(* IEC 61131-3 sources: RL_MAR/experiments/comparison/llm4plc/results/deepseek-ai-DeepSeek-V3.2_20260506_104945/20260506_124638, 3 files *)

(* ---- generated_code_iteration_0.st ---- *)
START_ST
FUNCTION_BLOCK CapsuleFillingMachineControl
VAR_INPUT
    CapsuleWeight : REAL;
    TargetWeight : REAL;
    CapsuleInPosition : BOOL;
    HopperEmpty : BOOL;
END_VAR
VAR_OUTPUT
    FeederMotor : BOOL;
    FillingMotor : BOOL;
    ConveyorMotor : BOOL;
    FillingInProgress : BOOL;
    ErrorFlag : BOOL;
    FillingTimeoutError : BOOL;
    CapsuleDetectionError : BOOL;
END_VAR
VAR
    state : INT;
    prevState : INT;
    fillingTimer : TON;
    conveyingTimer : TON;
    capsuleDetectionTimer : TON;
    tolerance : REAL := 0.1;
    conveyingTime : TIME := T#2s;
    fillingTimeout : TIME := T#10s;
    detectionTimeout : TIME := T#5s;
    pidController : PID;
    pidSetpoint : REAL;
    pidInput : REAL;
    pidOutput : REAL;
    pidKp : REAL := 1.0;
    pidKi : REAL := 0.1;
    pidKd : REAL := 0.05;
    manualReset : BOOL;
END_VAR

(* Safety Check - Immediate Override *)
IF HopperEmpty THEN
    FeederMotor := FALSE;
    FillingMotor := FALSE;
    ConveyorMotor := FALSE;
    FillingInProgress := FALSE;
    state := 4; (* ERROR state *)
    RETURN;
END_IF;

(* Weight Validation - Immediate Override *)
IF CapsuleWeight >= TargetWeight THEN
    FeederMotor := FALSE;
    FillingMotor := FALSE;
    ConveyorMotor := FALSE;
    FillingInProgress := FALSE;
    state := 4; (* ERROR state *)
    RETURN;
END_IF;

(* Main State Machine *)
CASE state OF
    0: (* IDLE *)
        FeederMotor := TRUE; (* Assumption: Feeder ON when not empty *)
        FillingMotor := FALSE;
        ConveyorMotor := FALSE;
        FillingInProgress := FALSE;
        ErrorFlag := FALSE;
        FillingTimeoutError := FALSE;
        CapsuleDetectionError := FALSE;

        capsuleDetectionTimer(IN:=FALSE, PT:=detectionTimeout);

        IF CapsuleInPosition AND (CapsuleWeight < TargetWeight) THEN
            state := 1; (* CONVEYING *)
            conveyingTimer(IN:=TRUE, PT:=conveyingTime);
        END_IF;

    1: (* CONVEYING *)
        FeederMotor := TRUE;
        FillingMotor := FALSE;
        ConveyorMotor := TRUE;
        FillingInProgress := FALSE;

        capsuleDetectionTimer(IN:=TRUE, PT:=detectionTimeout);

        (* Capsule Not Detected Error *)
        IF capsuleDetectionTimer.Q THEN
            CapsuleDetectionError := TRUE;
            ErrorFlag := TRUE;
            state := 4; (* ERROR *)
        END_IF;

        (* Transition to FILLING after conveying time *)
        conveyingTimer(IN:=TRUE, PT:=conveyingTime);
        IF conveyingTimer.Q THEN
            state := 2; (* FILLING *)
            fillingTimer(IN:=TRUE, PT:=fillingTimeout);
            pidSetpoint := TargetWeight;
        END_IF;

    2: (* FILLING *)
        FeederMotor := TRUE;
        FillingMotor := TRUE;
        ConveyorMotor := FALSE;
        FillingInProgress := TRUE;

        (* PID Control for Filling *)
        pidInput := CapsuleWeight;
        pidController(
            Setpoint:=pidSetpoint,
            Input:=pidInput,
            Kp:=pidKp,
            Ki:=pidKi,
            Kd:=pidKd,
            Output=>pidOutput
        );
        (* Note: In practice, pidOutput would control FillingMotor speed/valve *)

        (* Filling Timeout Error *)
        fillingTimer(IN:=TRUE, PT:=fillingTimeout);
        IF fillingTimer.Q THEN
            FillingTimeoutError := TRUE;
            ErrorFlag := TRUE;
            state := 4; (* ERROR *)
        END_IF;

        (* Weight Check with Tolerance *)
        IF CapsuleWeight >= (TargetWeight - tolerance) AND CapsuleWeight <= (TargetWeight + tolerance) THEN
            state := 3; (* CONVEYING_OUT *)
            conveyingTimer(IN:=TRUE, PT:=conveyingTime);
        END_IF;

    3: (* CONVEYING_OUT *)
        FeederMotor := TRUE;
        FillingMotor := FALSE;
        ConveyorMotor := TRUE;
        FillingInProgress := FALSE;

        (* Transition back to IDLE after conveying out *)
        conveyingTimer(IN:=TRUE, PT:=conveyingTime);
        IF conveyingTimer.Q THEN
            state := 0; (* IDLE *)
        END_IF;

    4: (* ERROR *)
        FeederMotor := FALSE;
        FillingMotor := FALSE;
        ConveyorMotor := FALSE;
        FillingInProgress := FALSE;

        (* Manual Reset Required *)
        IF manualReset AND NOT HopperEmpty AND (CapsuleWeight < TargetWeight) THEN
            state := 0; (* IDLE *)
            ErrorFlag := FALSE;
            FillingTimeoutError := FALSE;
            CapsuleDetectionError := FALSE;
        END_IF;

END_CASE;

(* Store previous state for debugging/monitoring *)
prevState := state;

END_FUNCTION_BLOCK
END_ST

(* ---- generated_code_iteration_1.st ---- *)
START_REASON
The validation feedback indicates that the CODESYS compiler validation failed due to an "未知的类型: 'PID'", which translates to "unknown type: 'PID'". This error occurs because the code uses a variable `pidController` of type `PID`, but the PID data type is not defined or declared in the current context. In Structured Text (ST) for CODESYS, `PID` is not a built-in primitive data type; it is typically a function block or a user-defined type that needs to be properly instantiated or defined. To fix this, I need to either:
1. Replace the PID controller with a custom implementation using basic arithmetic for proportional, integral, and derivative control, or
2. Use a standard PID function block if available in the CODESYS environment, but since the feedback doesn't specify available libraries, I'll assume a custom implementation is required for portability.

Given the original requirements, the PID controller is used for filling control based on weight. I can simplify this by using a basic proportional control or implement a custom PID logic. However, to keep the code functional and avoid undefined types, I'll remove the PID controller and replace it with a simpler control mechanism, such as turning the filling motor on/off based on weight comparison, since the feedback doesn't require complex PID tuning. This aligns with the state machine's purpose and avoids compiler errors.

Additionally, I'll ensure all variable declarations are correct and the code structure adheres to CODESYS standards, including proper use of `END_VAR` and maintaining the `FUNCTION_BLOCK` structure. The safety checks and state machine logic will be retained, but the PID-related variables and calls will be removed or replaced.
END_REASON

START_ST
FUNCTION_BLOCK CapsuleFillingMachineControl
VAR_INPUT
    CapsuleWeight : REAL;
    TargetWeight : REAL;
    CapsuleInPosition : BOOL;
    HopperEmpty : BOOL;
    manualReset : BOOL; (* Moved from VAR to VAR_INPUT for external control *)
END_VAR
VAR_OUTPUT
    FeederMotor : BOOL;
    FillingMotor : BOOL;
    ConveyorMotor : BOOL;
    FillingInProgress : BOOL;
    ErrorFlag : BOOL;
    FillingTimeoutError : BOOL;
    CapsuleDetectionError : BOOL;
END_VAR
VAR
    state : INT;
    prevState : INT;
    fillingTimer : TON;
    conveyingTimer : TON;
    capsuleDetectionTimer : TON;
    tolerance : REAL := 0.1;
    conveyingTime : TIME := T#2s;
    fillingTimeout : TIME := T#10s;
    detectionTimeout : TIME := T#5s;
    (* Removed PID controller and related variables to fix compiler error *)
END_VAR

(* Safety Check - Immediate Override: Stop all motors if hopper is empty *)
IF HopperEmpty THEN
    FeederMotor := FALSE;
    FillingMotor := FALSE;
    ConveyorMotor := FALSE;
    FillingInProgress := FALSE;
    state := 4; (* ERROR state *)
    RETURN;
END_IF;

(* Weight Validation - Immediate Override: Stop if capsule already at or above target weight *)
IF CapsuleWeight >= TargetWeight THEN
    FeederMotor := FALSE;
    FillingMotor := FALSE;
    ConveyorMotor := FALSE;
    FillingInProgress := FALSE;
    state := 4; (* ERROR state *)
    RETURN;
END_IF;

(* Main State Machine *)
CASE state OF
    0: (* IDLE: Waiting for capsule to be in position and under target weight *)
        FeederMotor := TRUE; (* Keep feeder on to supply material *)
        FillingMotor := FALSE;
        ConveyorMotor := FALSE;
        FillingInProgress := FALSE;
        ErrorFlag := FALSE;
        FillingTimeoutError := FALSE;
        CapsuleDetectionError := FALSE;

        capsuleDetectionTimer(IN:=FALSE, PT:=detectionTimeout); (* Reset detection timer *)

        IF CapsuleInPosition AND (CapsuleWeight < TargetWeight) THEN
            state := 1; (* Transition to CONVEYING *)
            conveyingTimer(IN:=TRUE, PT:=conveyingTime); (* Start conveying timer *)
        END_IF;

    1: (* CONVEYING: Moving capsule into filling position *)
        FeederMotor := TRUE;
        FillingMotor := FALSE;
        ConveyorMotor := TRUE; (* Conveyor motor on to move capsule *)
        FillingInProgress := FALSE;

        capsuleDetectionTimer(IN:=TRUE, PT:=detectionTimeout); (* Start detection timer *)

        (* Capsule Not Detected Error: If timer expires, capsule is missing *)
        IF capsuleDetectionTimer.Q THEN
            CapsuleDetectionError := TRUE;
            ErrorFlag := TRUE;
            state := 4; (* Transition to ERROR state *)
        END_IF;

        (* Transition to FILLING after conveying time elapses *)
        conveyingTimer(IN:=TRUE, PT:=conveyingTime);
        IF conveyingTimer.Q THEN
            state := 2; (* Transition to FILLING *)
            fillingTimer(IN:=TRUE, PT:=fillingTimeout); (* Start filling timeout timer *)
        END_IF;

    2: (* FILLING: Actively filling the capsule to target weight *)
        FeederMotor := TRUE;
        FillingMotor := TRUE; (* Filling motor on to dispense material *)
        ConveyorMotor := FALSE;
        FillingInProgress := TRUE;

        (* Simplified filling control: Motor stays on until weight reaches target with tolerance *)
        (* Removed PID controller to avoid compiler error; using direct weight comparison *)

        (* Filling Timeout Error: If timer expires, filling took too long *)
        fillingTimer(IN:=TRUE, PT:=fillingTimeout);
        IF fillingTimer.Q THEN
            FillingTimeoutError := TRUE;
            ErrorFlag := TRUE;
            state := 4; (* Transition to ERROR state *)
        END_IF;

        (* Weight Check with Tolerance: Stop filling when weight is within tolerance of target *)
        IF (CapsuleWeight >= (TargetWeight - tolerance)) AND (CapsuleWeight <= (TargetWeight + tolerance)) THEN
            state := 3; (* Transition to CONVEYING_OUT *)
            conveyingTimer(IN:=TRUE, PT:=conveyingTime); (* Start conveying timer for output *)
        END_IF;

    3: (* CONVEYING_OUT: Moving filled capsule out of the machine *)
        FeederMotor := TRUE;
        FillingMotor := FALSE;
        ConveyorMotor := TRUE; (* Conveyor motor on to move capsule out *)
        FillingInProgress := FALSE;

        (* Transition back to IDLE after conveying out time elapses *)
        conveyingTimer(IN:=TRUE, PT:=conveyingTime);
        IF conveyingTimer.Q THEN
            state := 0; (* Transition back to IDLE *)
        END_IF;

    4: (* ERROR: Error state, all motors stopped, requires manual reset *)
        FeederMotor := FALSE;
        FillingMotor := FALSE;
        ConveyorMotor := FALSE;
        FillingInProgress := FALSE;

        (* Manual Reset Required: Reset to IDLE if conditions are met and manualReset is TRUE *)
        IF manualReset AND (NOT HopperEmpty) AND (CapsuleWeight < TargetWeight) THEN
            state := 0; (* Transition to IDLE *)
            ErrorFlag := FALSE;
            FillingTimeoutError := FALSE;
            CapsuleDetectionError := FALSE;
        END_IF;

END_CASE;

(* Store previous state for debugging or monitoring purposes *)
prevState := state;

END_FUNCTION_BLOCK
END_ST

(* ---- generated_code_iteration_2.st ---- *)
START_REASON
The validation feedback indicates an encoding issue with the CODESYS compiler, specifically a 'gbk' codec can't decode byte 0xaa at position 105. This suggests there might be a non-ASCII character or encoding problem in the previous ST code submission. Since the error occurs during syntax check, it's likely that invisible or special characters were introduced. To fix this, I need to ensure the code uses only standard ASCII characters and proper Structured Text syntax. I'll rewrite the code from scratch, ensuring all characters are valid ASCII and the structure is correct. I'll maintain the FUNCTION_BLOCK structure, use proper variable declarations with END_VAR, and implement the state machine logic without PID controllers to avoid previous errors. The code will include safety checks, timers, and error handling as per requirements.
END_REASON

START_ST
FUNCTION_BLOCK CapsuleFillingMachineControl
VAR_INPUT
    CapsuleWeight : REAL;
    TargetWeight : REAL;
    CapsuleInPosition : BOOL;
    HopperEmpty : BOOL;
    manualReset : BOOL;
END_VAR
VAR_OUTPUT
    FeederMotor : BOOL;
    FillingMotor : BOOL;
    ConveyorMotor : BOOL;
    FillingInProgress : BOOL;
    ErrorFlag : BOOL;
    FillingTimeoutError : BOOL;
    CapsuleDetectionError : BOOL;
END_VAR
VAR
    state : INT;
    prevState : INT;
    fillingTimer : TON;
    conveyingTimer : TON;
    capsuleDetectionTimer : TON;
    tolerance : REAL := 0.1;
    conveyingTime : TIME := T#2s;
    fillingTimeout : TIME := T#10s;
    detectionTimeout : TIME := T#5s;
END_VAR

(* Safety Check - Immediate Override: Stop all motors if hopper is empty *)
IF HopperEmpty THEN
    FeederMotor := FALSE;
    FillingMotor := FALSE;
    ConveyorMotor := FALSE;
    FillingInProgress := FALSE;
    state := 4;
    RETURN;
END_IF;

(* Weight Validation - Immediate Override: Stop if capsule already at or above target weight *)
IF CapsuleWeight >= TargetWeight THEN
    FeederMotor := FALSE;
    FillingMotor := FALSE;
    ConveyorMotor := FALSE;
    FillingInProgress := FALSE;
    state := 4;
    RETURN;
END_IF;

(* Main State Machine *)
CASE state OF
    0: (* IDLE: Waiting for capsule to be in position and under target weight *)
        FeederMotor := TRUE;
        FillingMotor := FALSE;
        ConveyorMotor := FALSE;
        FillingInProgress := FALSE;
        ErrorFlag := FALSE;
        FillingTimeoutError := FALSE;
        CapsuleDetectionError := FALSE;

        capsuleDetectionTimer(IN:=FALSE, PT:=detectionTimeout);

        IF CapsuleInPosition AND (CapsuleWeight < TargetWeight) THEN
            state := 1;
            conveyingTimer(IN:=TRUE, PT:=conveyingTime);
        END_IF;

    1: (* CONVEYING: Moving capsule into filling position *)
        FeederMotor := TRUE;
        FillingMotor := FALSE;
        ConveyorMotor := TRUE;
        FillingInProgress := FALSE;

        capsuleDetectionTimer(IN:=TRUE, PT:=detectionTimeout);

        IF capsuleDetectionTimer.Q THEN
            CapsuleDetectionError := TRUE;
            ErrorFlag := TRUE;
            state := 4;
        END_IF;

        conveyingTimer(IN:=TRUE, PT:=conveyingTime);
        IF conveyingTimer.Q THEN
            state := 2;
            fillingTimer(IN:=TRUE, PT:=fillingTimeout);
        END_IF;

    2: (* FILLING: Actively filling the capsule to target weight *)
        FeederMotor := TRUE;
        FillingMotor := TRUE;
        ConveyorMotor := FALSE;
        FillingInProgress := TRUE;

        fillingTimer(IN:=TRUE, PT:=fillingTimeout);
        IF fillingTimer.Q THEN
            FillingTimeoutError := TRUE;
            ErrorFlag := TRUE;
            state := 4;
        END_IF;

        IF (CapsuleWeight >= (TargetWeight - tolerance)) AND (CapsuleWeight <= (TargetWeight + tolerance)) THEN
            state := 3;
            conveyingTimer(IN:=TRUE, PT:=conveyingTime);
        END_IF;

    3: (* CONVEYING_OUT: Moving filled capsule out of the machine *)
        FeederMotor := TRUE;
        FillingMotor := FALSE;
        ConveyorMotor := TRUE;
        FillingInProgress := FALSE;

        conveyingTimer(IN:=TRUE, PT:=conveyingTime);
        IF conveyingTimer.Q THEN
            state := 0;
        END_IF;

    4: (* ERROR: Error state, all motors stopped, requires manual reset *)
        FeederMotor := FALSE;
        FillingMotor := FALSE;
        ConveyorMotor := FALSE;
        FillingInProgress := FALSE;

        IF manualReset AND (NOT HopperEmpty) AND (CapsuleWeight < TargetWeight) THEN
            state := 0;
            ErrorFlag := FALSE;
            FillingTimeoutError := FALSE;
            CapsuleDetectionError := FALSE;
        END_IF;

END_CASE;

prevState := state;

END_FUNCTION_BLOCK
END_ST
